(* IEC 61131-3 sources: lc3-lib/I2C, 5 files *)

(* ---- Constants.iecst ---- *)
TYPE
	I2C_Constants : DINT (I2C_SLAVE := 1795); /* constant from the Linux kernel */
END_TYPE

(* ---- I2HAA.iecst ---- *)
FUNCTION I2C_I2HAA_write
	VAR_INPUT
		fd : DINT := -1;
		address : INT;
		values : ARRAY[0..4] OF UINT;
	END_VAR
	VAR
		bus_data : ARRAY[0..63] OF BYTE;
		cnt : USINT;
	END_VAR
	VAR CONSTANT
		num_channels : USINT := 5;
		num_bytes : USINT := 11;
	END_VAR;

	IF fd >= 0 THEN
		System_ioctl(fd := fd, request := I2C_Constants#I2C_SLAVE, data := address, ENO => ENO);
		IF ENO THEN
			bus_data[0] := 0;
			FOR cnt := 0 TO num_channels - 1 BY 1 DO
				bus_data[cnt * 2 + 1] := TO_BYTE(values[cnt] MOD 256);
				bus_data[cnt * 2 + 2] := TO_BYTE(values[cnt] / 256);
			END_FOR;

			ENO := System_write(fd := fd, count := num_bytes, data := bus_data) = num_bytes;
		END_IF;
	ELSE
		ENO := FALSE;
	END_IF;
END_FUNCTION

FUNCTION I2C_I2HAA_write_single
	VAR_INPUT
		fd : DINT := -1;
		address : INT;
		channel : USINT;
		value : UINT;
	END_VAR
	VAR
		bus_data : ARRAY[0..63] OF BYTE;
		checked_value : UINT := 1023;
	END_VAR
	VAR CONSTANT
		num_channels : USINT := 5;
		num_bytes : USINT := 3;
	END_VAR

	IF channel > num_channels - 1 THEN
		ENO := False;
		RETURN;
	END_IF;

	IF value < 1024 THEN
		checked_value := value;
	END_IF;

	IF fd >= 0 THEN
		System_ioctl(fd := fd, request := I2C_Constants#I2C_SLAVE, data := address, ENO => ENO);
		IF ENO THEN
			bus_data[0] := TO_BYTE(channel);
			bus_data[1] := TO_BYTE(checked_value MOD 256);
			bus_data[2] := TO_BYTE(checked_value / 256);
			ENO := System_write(fd := fd, count := num_bytes, data := bus_data) = num_bytes;
		END_IF;
	ELSE
		ENO := FALSE;
	END_IF;
END_FUNCTION

(* ---- I2HAE.iecst ---- *)
FUNCTION I2C_I2HAE_read
	VAR_INPUT
		fd : DINT := -1;
		address : INT;
	END_VAR
	VAR_OUTPUT
		values : ARRAY[0..4] OF UINT;
	END_VAR
	VAR
		bus_data : ARRAY[0..63] OF BYTE;
		num_bytes_read : DINT;
		cnt : USINT;
	END_VAR
	VAR CONSTANT
		num_channels : USINT := 5;
		num_bytes : USINT := 11;
	END_VAR

	IF fd >= 0 THEN
		System_ioctl(fd := fd, request := I2C_Constants#I2C_SLAVE, data := address, ENO => ENO);
		IF ENO THEN
			num_bytes_read := System_read(fd := fd, count := num_bytes, data := bus_data);
		END_IF;
		IF ENO AND num_bytes_read = num_bytes THEN
			FOR cnt := 0 TO num_channels - 1 BY 1 DO
				values[cnt] := TO_UINT(bus_data[1 + cnt * 2]) + TO_UINT(bus_data[2 + cnt * 2]) * 256;
			END_FOR;
		END_IF;
	ELSE
		ENO := FALSE;
	END_IF;
END_FUNCTION

(* ---- MAX7311.iecst ---- *)
FUNCTION I2C_MAX7311_write
	VAR_INPUT
		fd : DINT := -1;
		address : INT;
		pin_values : ARRAY[0..7] OF BOOL;
	END_VAR

	VAR
		num_bytes : DINT := -1; /* number of bytes written to bus device */
		cnt : INT := 0;
		data : ARRAY[0 .. 63] OF BYTE;
	END_VAR

	IF fd >= 0 THEN
		System_ioctl(fd := fd, request := I2C_Constants#I2C_SLAVE, data := address, ENO => ENO);
		IF ENO THEN
			data[0] := 16#06;
			FOR cnt := 0 TO 7 BY 1 DO
				data[1] := OR(data[1], SHL(pin_values[cnt], cnt));
			END_FOR;
			num_bytes := System_write(fd := fd, count := 2, data := data, ENO => ENO);
			IF num_bytes <> 2 THEN
				ENO := FALSE;
			END_IF;
		END_IF;
	ELSE
		ENO := FALSE;
	END_IF;
END_FUNCTION

(* ---- PCA9685.iecst ---- *)
FUNCTION PCA9685_selectPWMMode
	VAR_INPUT
		fd : DINT;
	END_VAR

	VAR
		mode1_val : USINT;

		/* constants: registers */
		mode1 : USINT := 16#00;
		mode2 : USINT := 16#01;

		/* constants: bits */
		allcall : USINT := 16#01;
		outdrv : USINT := 16#04;
		sleep : USINT := 16#10;
	END_VAR

	i2c_smbus_write_byte_data(fd := fd, command := mode2, value := outdrv);
	i2c_smbus_write_byte_data(fd := fd, command := mode1, value := allcall);
	/* TODO sleep */
	mode1_val := IAND(IN1 := TO_USINT(IN := i2c_smbus_read_byte_data(fd := fd, command := mode1)), IN2 := 16#FF);
	mode1_val := IAND(IN1 := mode1_val, IN2 := TO_USINT(NOT(IN := TO_BYTE(sleep))));
	i2c_smbus_write_byte_data(fd := fd, command := mode1, value := mode1_val);
	/* TODO sleep */
END_FUNCTION

FUNCTION PCA9685_setPWMFrequency
	VAR_INPUT
		fd : DINT;
		frequency : UDINT;
	END_VAR

	VAR
		prescaleval : LREAL := 25000000 /* MHz */;
		oldmode : USINT;
		newmode : USINT;

		/* constants */
		mode1 : USINT := 16#00;
		prescale : USINT := 16#FE;
	END_VAR

	prescaleval := prescaleval / 4096;
	prescaleval := prescaleval / frequency;
	prescaleval := prescaleval - 1;

	prescaleval := floor(prescaleval + 0.5);

	oldmode := TO_USINT(i2c_smbus_read_byte_data(fd := fd, command := mode1));
	newmode := IOR(IN1 := IAND(IN1 := oldmode, IN2 := 16#7f), IN2 := 16#10);

	i2c_smbus_write_byte_data(fd := fd, command := mode1, value := newmode);
	i2c_smbus_write_byte_data(fd := fd, command := prescale, value := TO_USINT(prescaleval));
	i2c_smbus_write_byte_data(fd := fd, command := mode1, value := oldmode);
	i2c_smbus_write_byte_data(fd := fd, command := mode1, value := IOR(IN1 := oldmode, IN2 := 16#80));
END_FUNCTION

FUNCTION PCA9685_setAllPWM
	VAR_INPUT
		fd : DINT;
		on_value : UINT;
		off_value : UINT;
	END_VAR

	VAR
		ALL_LED_ON_L : USINT := 16#FA;
		ALL_LED_ON_H : USINT := 16#FB;
		ALL_LED_OFF_L : USINT := 16#FC;
		ALL_LED_OFF_H : USINT := 16#FD;
	END_VAR

	i2c_smbus_write_byte_data(fd := fd, command := ALL_LED_ON_L, value := TO_USINT(IAND(IN1 := on_value, IN2 := 16#FF)));
	i2c_smbus_write_byte_data(fd := fd, command := ALL_LED_ON_H, value := TO_USINT(SAR(IN := on_value, N := 8)));
	i2c_smbus_write_byte_data(fd := fd, command := ALL_LED_OFF_L, value := TO_USINT(IAND(IN1 := off_value, IN2 := 16#FF)));
	i2c_smbus_write_byte_data(fd := fd, command := ALL_LED_OFF_H, value := TO_USINT(SAR(IN := off_value, N := 8)));
END_FUNCTION

FUNCTION setPWM
	VAR_INPUT
		fd : DINT;
		channel : USINT;
		on_value : UINT;
		off_value : UINT;
	END_VAR

	VAR
		LED0_ON_L : USINT := 16#06;
		LED0_ON_H : USINT := 16#07;
		LED0_OFF_L : USINT := 16#08;
		LED0_OFF_H : USINT := 16#09;
	END_VAR

	i2c_smbus_write_byte_data(fd := fd, command := LED0_ON_L + 4 * channel, value := TO_USINT(IAND(IN1 := on_value, IN2 := 16#FF)));
	i2c_smbus_write_byte_data(fd := fd, command := LED0_ON_H + 4 * channel, value := TO_USINT(SAR(IN := on_value, N := 8)));
	i2c_smbus_write_byte_data(fd := fd, command := LED0_OFF_L + 4 * channel, value := TO_USINT(IAND(IN1 := off_value, IN2 := 16#FF)));
	i2c_smbus_write_byte_data(fd := fd, command := LED0_OFF_H + 4 * channel, value := TO_USINT(SAR(IN := off_value, N := 8)));
END_FUNCTION
